(* PLC project mclamping, Dassault Systèmes ControlBuild 2024x *)
(* stored: creationDateTime 2023-10-03T11:13:46-01:00 *)

PROGRAM drill.mclamping
  VAR_INPUT
    acknowledgePB : BOOL := false;
  END_VAR
  VAR_INPUT
    autoMode : BOOL := false;
    manualMode : BOOL := false;
  END_VAR
  VAR_INPUT
    releasing : BOOL := false;
    clamping : BOOL := false;
  END_VAR
  VAR_OUTPUT
    clampingOK : BOOL := false;
    releasingOK : BOOL := false;
    clampingFault : DINT := 0;
  END_VAR

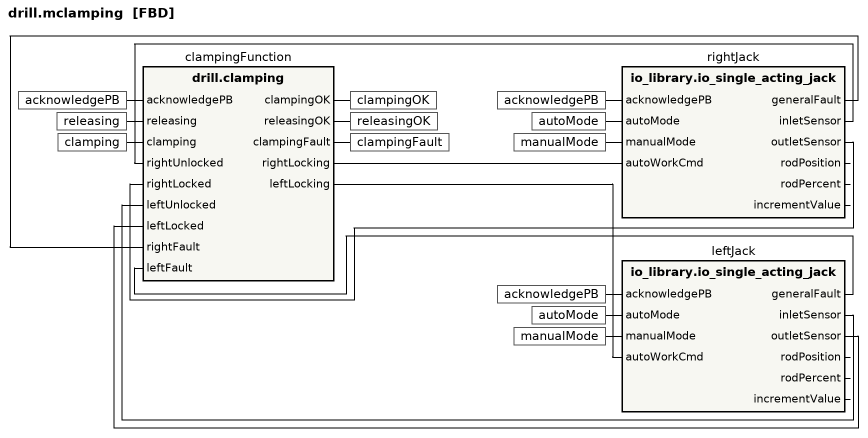
(* FBD diagram, written out as Structured Text *)
rightJack(acknowledgePB := acknowledgePB, autoMode := autoMode, manualMode := manualMode, autoWorkCmd := clampingFunction.rightLocking);
leftJack(acknowledgePB := acknowledgePB, autoMode := autoMode, manualMode := manualMode, autoWorkCmd := clampingFunction.leftLocking);
clampingFunction(acknowledgePB := acknowledgePB, releasing := releasing, clamping := clamping, rightUnlocked := rightJack.inletSensor, rightLocked := rightJack.outletSensor, leftUnlocked := leftJack.inletSensor, leftLocked := leftJack.outletSensor, rightFault := rightJack.generalFault, leftFault := leftJack.generalFault);
clampingOK := clampingFunction.clampingOK;
releasingOK := clampingFunction.releasingOK;
clampingFault := clampingFunction.clampingFault;
END_PROGRAM
